TYPE ST_AdjustmentPositionConfig :
STRUCT
    stReady : ST_Point3D;
    stWork : ST_Point3D;
END_STRUCT
END_TYPE

(* stored: Version 1.1.0.1, ProductVersion 3.1.4026.20
   DUT ST_AdjustmentPositionConfig: Id {3868465d-c7c9-4806-9fdb-9de513f64122} *)
